// TIA Portal V21 export
DATA_BLOCK "L"   // DB187
{ S7_Optimized_Access := 'TRUE' }
// stored: MemoryReserve 100
   VAR RETAIN
      "DATE" : USInt;
      MONTH : USInt;
      YEAR : UInt;
      LO : Int;
      FIRMAWARE : Bool;
      "CIRON PRINT" : Bool;
      "STD VACUUM DIS" : Bool;
   END_VAR
BEGIN
END_DATA_BLOCK
